{attribute 'qualified_only'}
{attribute 'strict'}
TYPE ePiston :
(
	off := 0,
	running,
	fwd,
	bkw,
	error
);
END_TYPE

(* stored: Version 1.1.0.1, ProductVersion 3.1.4022.18
   DUT ePiston: Id {f2cac472-bac7-4569-834a-a6e1f06df81d} *)
